// TIA Portal V19 export
DATA_BLOCK "TSEND_DI"   // DB366
// stored: AutoNumber false, InstanceOfName TSEND, OfSystemLibElement TSEND, OfSystemLibVersion 4.0
"TSEND"
   // VAR_INPUT
   //    REQ : Bool := TRUE;
   //    ID : CONN_OUC := 16#0002;
   //    LEN : UDInt := 30;
   // END_VAR
   // VAR_OUTPUT
   //    DONE : Bool := TRUE;
   //    BUSY : Bool := FALSE;
   //    ERROR : Bool := FALSE;
   //    STATUS : Word := 16#0000;
   // END_VAR
   // VAR_IN_OUT
   //    DATA : Variant;
   //    ADDR : Variant;
   // END_VAR
BEGIN
END_DATA_BLOCK
